FUNCTION_BLOCK WagoMaster (* Service Interface Function Block Type *)
  (* Standard: 61499-2; Description: Copyright (c) 2018 fortiss GmbH This program and the accompanying materials are made available under the terms of the Eclipse Public License 2.0 which is available at https://www.eclipse.org/legal/epl-2.0/ SPDX-License-Identifier: EPL-2.0 *)
  (* Version 1.0, 2018-12-05, Jose Cabral *)
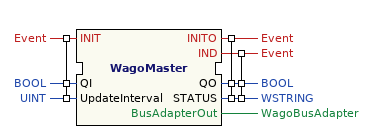
  EVENT_INPUT
    INIT WITH QI, UpdateInterval; (* Service Initialization *)
  END_EVENT
  EVENT_OUTPUT
    INITO WITH QO, STATUS; (* Initialization Confirm *)
    IND WITH STATUS, QO; (* Indication from Resource *)
  END_EVENT
  VAR_INPUT
    QI : BOOL; (* Event Input Qualifier *)
    UpdateInterval : UINT;
  END_VAR
  VAR_OUTPUT
    QO : BOOL; (* Event Output Qualifier *)
    STATUS : WSTRING; (* Service Status *)
  END_VAR
  PLUGS
    BusAdapterOut : WagoBusAdapter;
  END_PLUGS
END_FUNCTION_BLOCK
